// TIA Portal V19 export
TYPE "LAF_typeXyzhandlingEm4ParametersInterface"
// stored: Access Published
   STRUCT
      configuration : "LAF_typeXyzhandlingEm4Parameters";
      commands : "LBC_typeInterfaceCommands";
      monitoring { S7_SetPoint := 'True'} : "LAF_typeXyzhandlingEm4ProcessValues";
   END_STRUCT;
END_TYPE
